FUNCTION_BLOCK FindRed
VAR_INPUT 
	hr 				: HRESULT;
	ipImageIn		: ITcVnImage;
	aLowerRedBottom	: TcVnVector4_LREAL;
	aLowerRedTop		: TcVnVector4_LREAL;
	aUpperRedBottom	: TcVnVector4_LREAL;
	aUpperRedTop		: TcVnVector4_LREAL;
END_VAR
VAR_OUTPUT
	ipImageOut		: ITcVnImage; //Returns a Grey image of where the red is
END_VAR
VAR
	ipImageColorMap_Red: ITcVnImage;
	ipImageColorMap_Red2: ITcVnImage;
	ipImageColorMap_Red3: ITcVnImage;
END_VAR
VAR_IN_OUT
	
END_VAR

//Creating first mask
hr := F_VN_CheckColorRange(ipImageIn, ipImageColorMap_Red,aLowerRedBottom,aLowerRedTop,hr);
//creating second mask
hr := F_VN_CheckColorRange(ipImageIn, ipImageColorMap_Red2,aUpperRedBottom,aUpperRedTop,hr);
//Adding masks together
hr := F_VN_BitwiseOrImages(ipImageColorMap_Red,ipImageColorMap_Red2,ipImageColorMap_Red3,hr);

END_FUNCTION_BLOCK

(* stored: Version 1.1.0.1, ProductVersion 3.1.4024.12
   POU FindRed: Id {32f2a2dc-54a1-476d-862d-3227091e7746}, SpecialFunc None *)
